{attribute 'qualified_only' := ''}
VAR_GLOBAL CONSTANT
	NUMOFSUBSCRIBERS: INT := 10;
END_VAR

(* stored: Version 1.1.0.1
   GVL Gl1: Id {116ab916-0d90-45c1-b134-6a47a1442507} *)
